FUNCTION_BLOCK SERVICE_INFO_JSON_SERIALIZE (* Composite Function Block Type *)
  (* Standard: 61499-2 *)
  (* Version 0.0, 12/30/2022, brink, Flexbridge AB, template *)
  PACKAGE UAO.Hackathon;
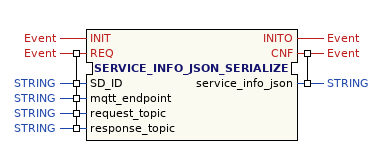
  EVENT_INPUT
    INIT;
    REQ WITH SD_ID, mqtt_endpoint, request_topic, response_topic;
  END_EVENT
  EVENT_OUTPUT
    INITO;
    CNF WITH service_info_json; (* Execution Confirmation *)
  END_EVENT
  VAR_INPUT
    SD_ID : STRING;
    mqtt_endpoint : STRING;
    request_topic : STRING;
    response_topic : STRING;
  END_VAR
  VAR_OUTPUT
    service_info_json : STRING;
  END_VAR
  FBS
    FB3 : JSON_FORMAT_12F3DFA5AB90F4A4(format := '{service_info:{SD_ID:"%s",mqtt_endpoint:"%s",mqtt_topic:"%s"}}'); {SET_ATTRIBUTE(Configuration.GenericFBType.InterfaceParams, Runtime.Base#CNT:=3;value${CNT$}:STRING,STRING,STRING)}
    FB4 : ADD_REMOVE_SLASH;
    FB5 : JSON_FORMAT_12F3DFA5AB90F4A4(format := '{service_info:{SD_ID:"%s",mqtt_endpoint:"%s",mqtt_topic:"%s"}}'); {SET_ATTRIBUTE(Configuration.GenericFBType.InterfaceParams, Runtime.Base#CNT:=3;value${CNT$}:STRING,STRING,STRING)}
    FB6 : ADD_REMOVE_SLASH;
    FB7 : JSON_FORMAT_12F3DFA5AB90F4A4(format := '{service_info:{SD_ID:"%s",mqtt_endpoint:"%s",mqtt_topic:"%s"}}'); {SET_ATTRIBUTE(Configuration.GenericFBType.InterfaceParams, Runtime.Base#CNT:=3;value${CNT$}:STRING,STRING,STRING)}
    FB8 : JSON_FORMAT_12F3DFA5AB90F4A4(format := '{service_info:{SD_ID:"%s",mqtt_endpoint:"%s",mqtt_topic:"%s"}}'); {SET_ATTRIBUTE(Configuration.GenericFBType.InterfaceParams, Runtime.Base#CNT:=3;value${CNT$}:STRING,STRING,STRING)}
    FB1 : JSON_FORMAT_12EFF7739F51B62A(format := '{service_info:{SD_ID:"%s",mqtt_endpoint:"%s",request_topic:"%s",response_topic:"%s"}}'); {SET_ATTRIBUTE(Configuration.GenericFBType.InterfaceParams, Runtime.Base#CNT:=4;value${CNT$}:STRING,STRING,STRING,STRING)}
    FB2 : ADD_REMOVE_SLASH;
  END_FBS
  EVENT_CONNECTIONS
    FB2.ADD_SLASHO TO CNF;
    INIT TO FB1.SET_FORMAT;
    REQ TO FB1.REQ;
    FB1.SET_FORMAT_CNF TO INITO;
    FB1.CNF TO FB2.ADD_SLASH;
  END_CONNECTIONS
  DATA_CONNECTIONS
    FB2.OutputString TO service_info_json;
    SD_ID TO FB1.value1;
    mqtt_endpoint TO FB1.value2;
    request_topic TO FB1.value3;
    FB1.payload TO FB2.InputString;
    response_topic TO FB1.value4;
  END_CONNECTIONS
END_FUNCTION_BLOCK
